{attribute 'OPC.UA.DA' := '1'}
{attribute 'OPC.UA.DA.StructuredType' := '1'}
TYPE CustomMsg :
STRUCT	
	Id : EPowerIlluminationFlow;
	Custom : STRING(255);
END_STRUCT
END_TYPE

(* stored: Version 1.1.0.1, ProductVersion 3.1.4024.3
   DUT CustomMsg: Id {53e2072b-f459-4123-84a8-e6fdcd5741c0} *)
